(*
Struct inside ExampleFolder.
*)
TYPE ST_ExampleFolder_Struct :
STRUCT
END_STRUCT
END_TYPE

(* stored: Version 1.1.0.1, ProductVersion 3.1.4024.11
   DUT ST_ExampleFolder_Struct: Id {f56a56da-26d1-4423-8d1c-2a4ffe32178d} *)
